{attribute 'qualified_only'}
VAR_GLOBAL CONSTANT
	AXIS_NAME_SIZE: DINT := 9;
	FAULT_STRING_SIZE: DINT := 19;
	FAULT_ARRAY_SIZE: DINT := 10;
	STATUS_STRING_SIZE: DINT := 19;
	ANALOG_ARRAY_SIZE : DINT := 20;
END_VAR

(* stored: Version 1.1.0.1, ProductVersion 3.1.4022.12
   GVL CT: Id {ab1f46a4-6d6b-4d22-a611-752d5f043f1a} *)
